// TIA Portal V20 export
DATA_BLOCK "IDB_DataMan262"   // DB40
// stored: InstanceOfName Global.DataMan262, InstanceOfType FB, Namespace Global
"Global.DataMan262"
   // VAR_INPUT
   //    TriggerSignal : Bool;
   //    ContinuousGetResults : Bool;
   //    "Dataman-Results Available" : Bool;
   //    "Dataman-TriggerReady" : Bool;
   //    "Dataman-TriggerAck" : Bool;
   //    "Dataman-Train Focus Ack" : Bool;
   //    "Dataman-Train Match String Ack" : Bool;
   //    "Dataman-Execute DMCC Ack" : Bool;
   //    "Dataman-Set Match String Ack" : Bool;
   //    "Dataman-ResultID" : Int;
   //    "Dataman-Result Code" : Int;
   //    "Dataman-Result Length" : Int;
   //    "Result Data" : "Global.BarCode";
   // END_VAR
   // VAR_OUTPUT
   //    "Dataman-UserData Length" : Word;
   //    "Dataman-UserData Option" : Word;
   //    "User Data" : "Global.BarCode";
   // END_VAR
   // VAR_IN_OUT
   //    "Dataman-TriggerEnable" : Bool;
   //    "Dataman-Trigger" : Bool;
   //    "Dataman-ResultsAck" : Bool;
   //    "Dataman-Train Focus" : Bool;
   //    "Dataman-Train Match String" : Bool;
   //    "Dataman-Execute DMCC" : Bool;
   //    "Dataman-Set Match String" : Bool;
   // END_VAR
   // VAR
   //    "Result Pending" : Bool;
   //    "Latest Results" : Struct
   //       ID : Int;
   //       Flags : Int;
   //       Length : Int;
   //       Value : Array[0..63] of Byte;
   //    END_STRUCT;
   //    "Train Focus" : Bool;
   //    "Train MatchString" : Bool;
   //    "Execute DMCC" : Bool;
   //    "Set Match String" : Bool;
   //    "String" : String[64];
   //    "Match String" : Array[0..63] of Byte;
   //    "Char" : Array[0..63] of Byte;
   //    Ret_val_1 { ExternalAccessible := 'False'; ExternalVisible := 'False'; ExternalWritable := 'False'} : Byte;
   //    R_TRIG_SimpleRead { S7_SetPoint := 'True'} : R_TRIG;
   //    R_TRIG_TrainFocus { S7_SetPoint := 'True'} : R_TRIG;
   //    "R_TRIG_Train MatchString" { S7_SetPoint := 'True'} : R_TRIG;
   //    R_TRIG_ExcuteDMCC { S7_SetPoint := 'True'} : R_TRIG;
   //    R_TRIG_SetMatchString { S7_SetPoint := 'True'} : R_TRIG;
   //    HoldTrigger { S7_SetPoint := 'True'} : Bool;
   //    HoldTrainFocus : Bool;
   //    HoldTrainMatchString : Bool;
   //    HoldDMCCExcute : Bool;
   //    HoldSetMatchString : Bool;
   // END_VAR
BEGIN
END_DATA_BLOCK
